(* Logix 5000 project; controller MecaB_Project vendor 1 type 14 code 155 rev 28.11; software revision 28.00 *)

TASK MainTask (continuous, watchdog 500 ms) : MainProgram

MODULES
   Local : vendor 1 type 14 code 155 (PointIO 0, rev 28.11)
      PR0_IP21 : vendor 1 type 37 code 27 (Ethernet 192.168.1.21, rev 1.1, MotionSync RPI 1 ms, MotionDiagnostics RPI 1 ms)
      PR0_IP22 : vendor 1 type 37 code 27 (Ethernet 192.168.1.22, rev 1.1, MotionDiagnostics RPI 1 ms, MotionSync RPI 1 ms)
      Discrete_IO : Embedded (PointIO 1, rev 28.11, Output RPI 20 ms)
END_MODULES

VAR_GLOBAL   (* controller tags *)
   Axis21 : AXIS_CIP_DRIVE;
   Axis21_MAFR : MOTION_INSTRUCTION := (FLAGS := 33554432);
   Axis21_MAM : MOTION_INSTRUCTION := (FLAGS := 301989888, ER := 1, ERR := 5);
   Axis21_MASR : MOTION_INSTRUCTION := (FLAGS := 33554432);
   Axis21_MSF : MOTION_INSTRUCTION := (FLAGS := 33554432);
   Axis21_MSO : MOTION_INSTRUCTION := (FLAGS := 301989888, ER := 1, ERR := 82);
   Axis21_Off : BOOL;
   Axis21_OffLamp : BOOL;
   Axis21_On : BOOL;
   Axis21_OnLamp : BOOL := 1;
   Axis21_Pos : REAL := 21.0;
   Axis21_SP : REAL;
   Axis22 : AXIS_CIP_DRIVE;
   Axis22_MAFR : MOTION_INSTRUCTION := (FLAGS := 33554432);
   Axis22_MAM : MOTION_INSTRUCTION := (FLAGS := 301989888, ER := 1, ERR := 5);
   Axis22_MASR : MOTION_INSTRUCTION := (FLAGS := 33554432);
   Axis22_MSF : MOTION_INSTRUCTION := (FLAGS := 33554432);
   Axis22_MSO : MOTION_INSTRUCTION := (FLAGS := 301989888, ER := 1, ERR := 82);
   Axis22_Off : BOOL;
   Axis22_OffLamp : BOOL;
   Axis22_On : BOOL;
   Axis22_OnLamp : BOOL := 1;
   Axis22_Pos : REAL := 51.0;
   Axis_Group : MOTION_GROUP;
   Axis_MotionStart : BOOL;
   Axis_Off : BOOL;
   Axis_On : BOOL;
   Axis_PositionRst : BOOL;
   Axis_Rst : BOOL;
   Axis_SP : REAL;
   LED_Timer : TIMER := (PRE := 500);
   LEDB : ALIAS FOR Local:1:O.Data.4;
   LEDB_OFF : BOOL;
   LEDB_ON : BOOL;
   LEDB_START : BOOL;
   LEDB_TON : BOOL;
   LEDG : ALIAS FOR Local:1:O.Data.3;
   LEDG_OFF : BOOL;
   LEDG_ON : BOOL;
   LEDG_START : BOOL;
   LEDG_TON : BOOL;
   LEDR : ALIAS FOR Local:1:O.Data.2;
   LEDR_OFF : BOOL;
   LEDR_ON : BOOL;
   LEDR_TON : BOOL;
   LEDRGB_OFF : BOOL;
   LEDRGB_ON : BOOL;
   LEDRGB_START : BOOL;
   MOVE : DINT;
   On21 : BOOL;
   On22 : BOOL;
   RUN : DINT := 999;
   Servo_On21 : ALIAS FOR Local:1:O.Data.0;
   Servo_On22 : ALIAS FOR Local:1:O.Data.1;
   TIME_LED : TIMER := (PRE := 500);
   TIME_LEDB : TIMER := (PRE := 500);
   TIME_LEDG : TIMER := (PRE := 500);
END_VAR

PROGRAM MainProgram   (* main routine MainRoutine *)

ROUTINE Axis21_Program   (* ladder *)
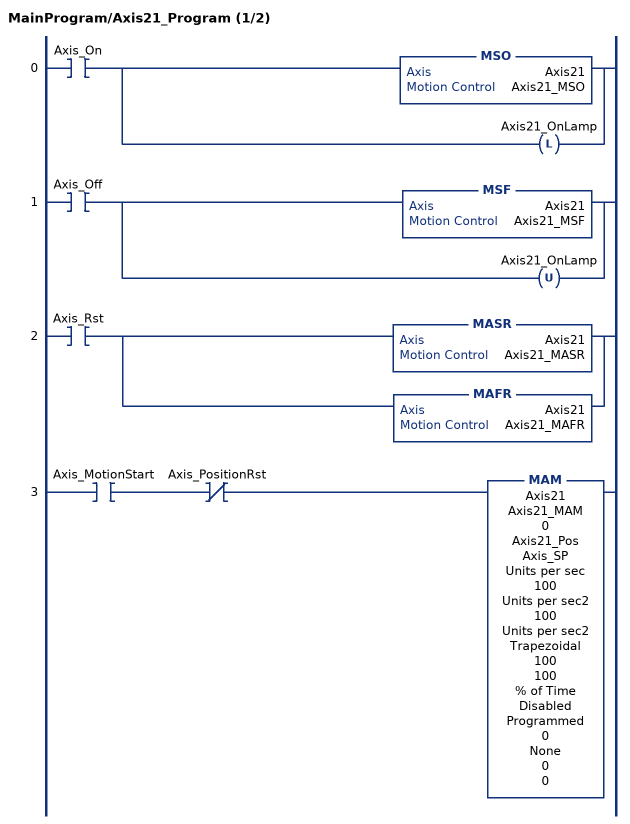
   0: XIC(Axis_On)[MSO(Axis21,Axis21_MSO) ,OTL(Axis21_OnLamp) ];
   1: XIC(Axis_Off)[MSF(Axis21,Axis21_MSF) ,OTU(Axis21_OnLamp) ];
   2: XIC(Axis_Rst)[MASR(Axis21,Axis21_MASR) ,MAFR(Axis21,Axis21_MAFR) ];
   3: XIC(Axis_MotionStart)XIO(Axis_PositionRst)MAM(Axis21,Axis21_MAM,0,Axis21_Pos,Axis_SP,Units per sec,100,Units per sec2,100,Units per sec2,Trapezoidal,100,100,% of Time,Disabled,Programmed,0,None,0,0);
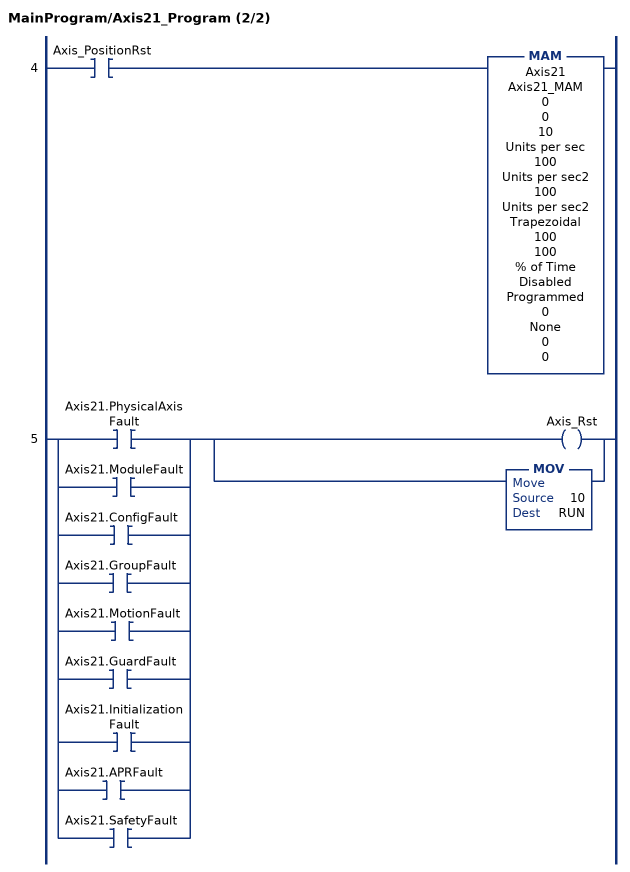
   4: XIC(Axis_PositionRst)MAM(Axis21,Axis21_MAM,0,0,10,Units per sec,100,Units per sec2,100,Units per sec2,Trapezoidal,100,100,% of Time,Disabled,Programmed,0,None,0,0);
   5: [XIC(Axis21.PhysicalAxisFault) ,XIC(Axis21.ModuleFault) ,XIC(Axis21.ConfigFault) ,XIC(Axis21.GroupFault) ,XIC(Axis21.MotionFault) ,XIC(Axis21.GuardFault) ,XIC(Axis21.InitializationFault) ,XIC(Axis21.APRFault) ,XIC(Axis21.SafetyFault) ][OTE(Axis_Rst) ,MOV(10,RUN) ];
END_ROUTINE

ROUTINE Axis22_Program   (* ladder *)
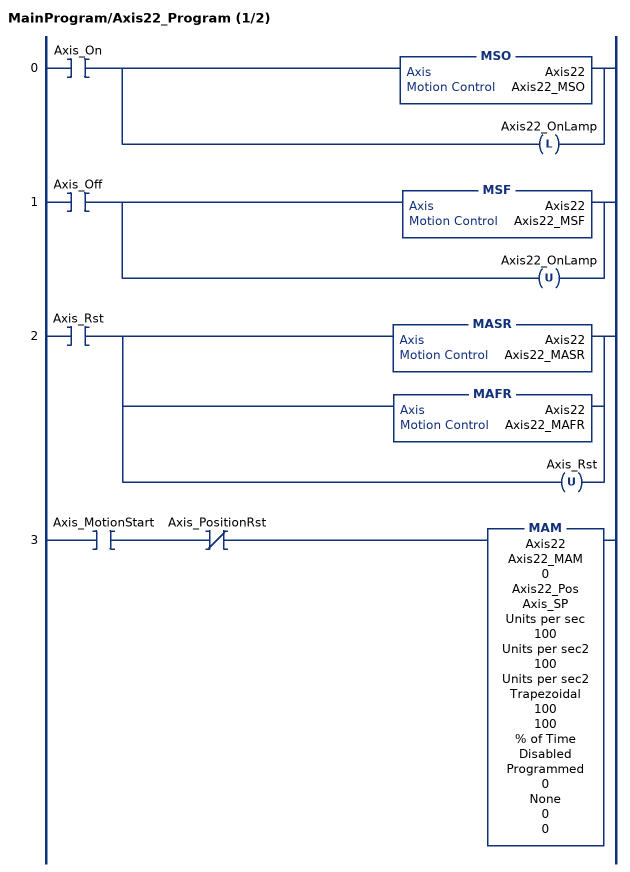
   0: XIC(Axis_On)[MSO(Axis22,Axis22_MSO) ,OTL(Axis22_OnLamp) ];
   1: XIC(Axis_Off)[MSF(Axis22,Axis22_MSF) ,OTU(Axis22_OnLamp) ];
   2: XIC(Axis_Rst)[[MASR(Axis22,Axis22_MASR) ,MAFR(Axis22,Axis22_MAFR) ] ,OTU(Axis_Rst) ];
   3: XIC(Axis_MotionStart)XIO(Axis_PositionRst)MAM(Axis22,Axis22_MAM,0,Axis22_Pos,Axis_SP,Units per sec,100,Units per sec2,100,Units per sec2,Trapezoidal,100,100,% of Time,Disabled,Programmed,0,None,0,0);
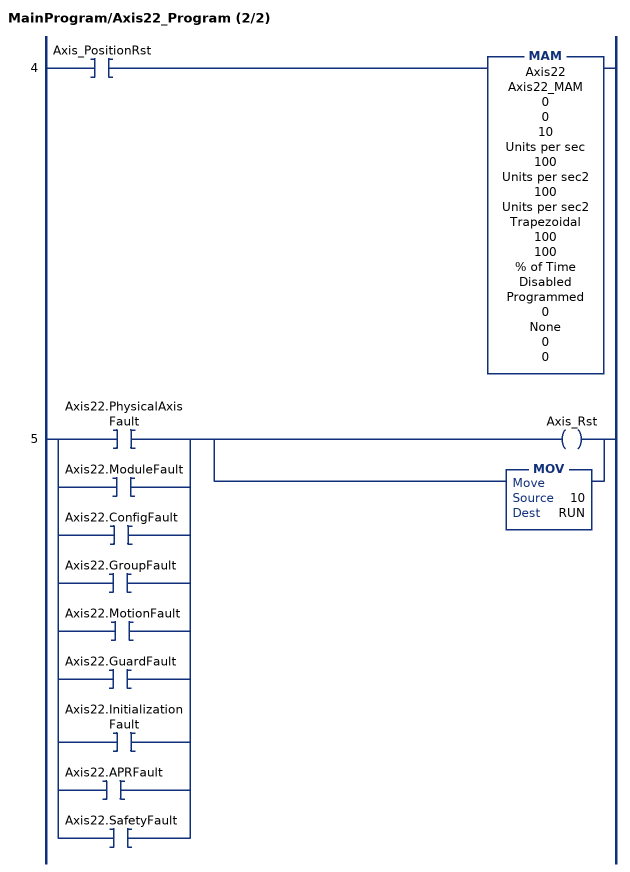
   4: XIC(Axis_PositionRst)MAM(Axis22,Axis22_MAM,0,0,10,Units per sec,100,Units per sec2,100,Units per sec2,Trapezoidal,100,100,% of Time,Disabled,Programmed,0,None,0,0);
   5: [XIC(Axis22.PhysicalAxisFault) ,XIC(Axis22.ModuleFault) ,XIC(Axis22.ConfigFault) ,XIC(Axis22.GroupFault) ,XIC(Axis22.MotionFault) ,XIC(Axis22.GuardFault) ,XIC(Axis22.InitializationFault) ,XIC(Axis22.APRFault) ,XIC(Axis22.SafetyFault) ][OTE(Axis_Rst) ,MOV(10,RUN) ];
END_ROUTINE

ROUTINE MainRoutine   (* ladder *)
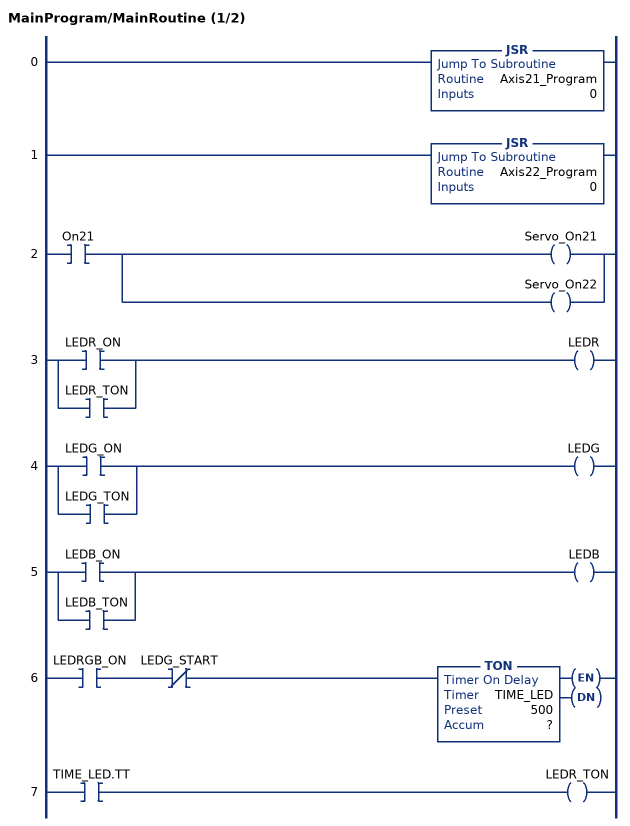
   0: JSR(Axis21_Program,0);
   1: JSR(Axis22_Program,0);
   2: XIC(On21)[OTE(Servo_On21) ,OTE(Servo_On22) ];
   3: [XIC(LEDR_ON) ,XIC(LEDR_TON) ]OTE(LEDR);
   4: [XIC(LEDG_ON) ,XIC(LEDG_TON) ]OTE(LEDG);
   5: [XIC(LEDB_ON) ,XIC(LEDB_TON) ]OTE(LEDB);
   6: XIC(LEDRGB_ON)XIO(LEDG_START)TON(TIME_LED,?,?);
   7: XIC(TIME_LED.TT)OTE(LEDR_TON);
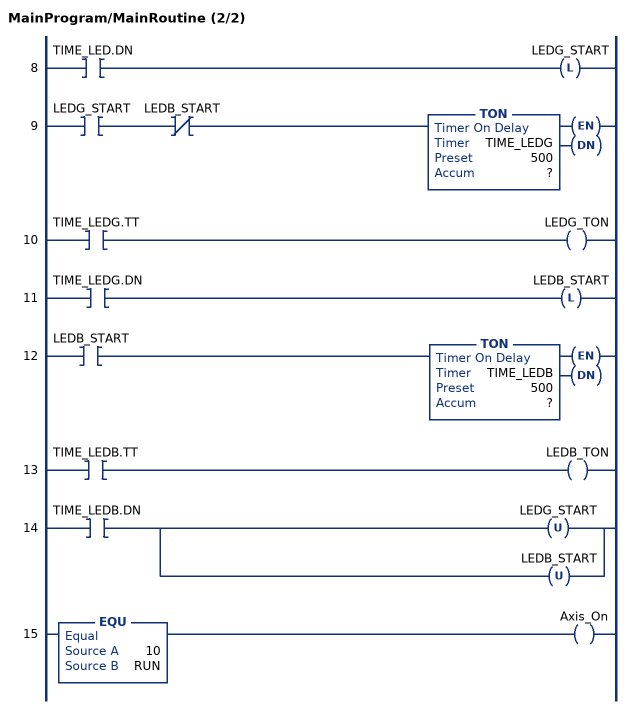
   8: XIC(TIME_LED.DN)OTL(LEDG_START);
   9: XIC(LEDG_START)XIO(LEDB_START)TON(TIME_LEDG,?,?);
   10: XIC(TIME_LEDG.TT)OTE(LEDG_TON);
   11: XIC(TIME_LEDG.DN)OTL(LEDB_START);
   12: XIC(LEDB_START)TON(TIME_LEDB,?,?);
   13: XIC(TIME_LEDB.TT)OTE(LEDB_TON);
   14: XIC(TIME_LEDB.DN)[OTU(LEDG_START) ,OTU(LEDB_START) ];
   15: EQU(10,RUN)OTE(Axis_On);
END_ROUTINE
END_PROGRAM
